// TIA Portal V19 export
FUNCTION_BLOCK "ButtonsSafe_LB211"   // FB167, LAD
TITLE = LB211 SAFE BUTTONS (@Rollformer) used for feed Area 02 material
// stored: MemoryReserve 100, SetENOAutomatically false
   VAR_INPUT
      Reset_OthersPBs_Activation_IN : Bool := FALSE;
   END_VAR
   VAR_OUTPUT
      Reset_OthersPBs_Activation_OUT : Bool;
   END_VAR
   VAR
      SelectionIs_Bwd : Bool;
      SelectionIs_Fwd : Bool;
      Pb_PEAux : Bool;
      PB : Struct
         ResetAlarms : Bool;
         Rollformer_Bwd : Bool;
         Rollformer_Fwd : Bool;
      END_STRUCT;
   END_VAR
   VAR_TEMP
      EnablingSwitch : Bool;
      Pb_PositiveEdge : Bool;
   END_VAR
   VAR_TEMP   // added for the SCL form of the ladder/FBD networks
      _w1 : Bool;
   END_VAR
BEGIN

REGION Network 1: Enabling switch positive edge
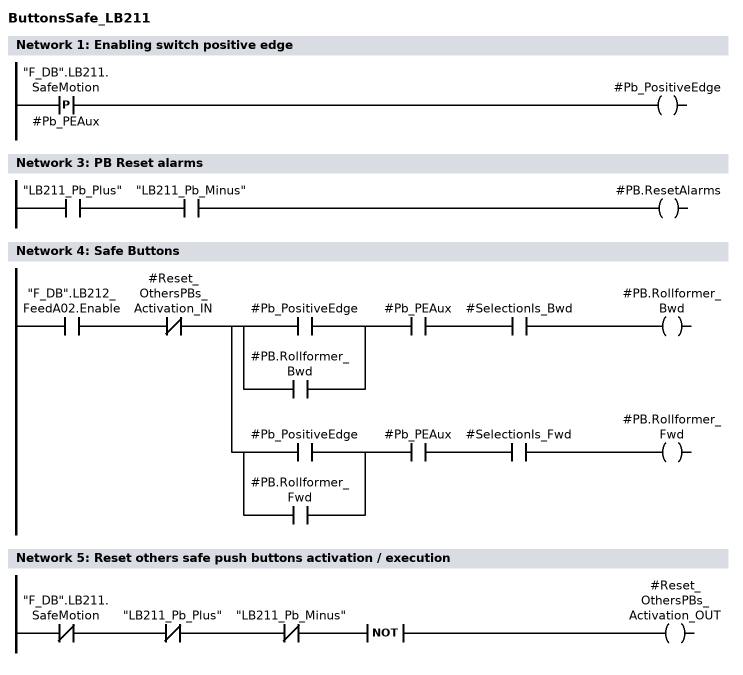
   RUNG wire#powerrail
      P_Contact(operand := "F_DB".LB211.SafeMotion, bit := #Pb_PEAux)
      Coil( #Pb_PositiveEdge )
   END_RUNG
   // the same network as SCL:
   #_w1 := "F_DB".LB211.SafeMotion AND NOT #Pb_PEAux;   // rising edge of "F_DB".LB211.SafeMotion
   #Pb_PEAux := "F_DB".LB211.SafeMotion;
   #Pb_PositiveEdge := #_w1;
END_REGION

REGION Network 2 (SCL): Selection of direction

   IF "LB211_Pb_Plus" AND  "LB211_Pb_Minus" THEN
       #SelectionIs_Fwd := FALSE;
       #SelectionIs_Bwd := FALSE;

   ELSIF "F_DB".LB211.SafeMotion THEN
       ;

   ELSIF "LB211_Pb_Plus" AND NOT "LB211_Pb_Minus"  THEN
       #SelectionIs_Fwd := TRUE;
       #SelectionIs_Bwd := FALSE;

   ELSIF "LB211_Pb_Minus" AND NOT "LB211_Pb_Plus" THEN
       #SelectionIs_Bwd := TRUE;       
       #SelectionIs_Fwd := FALSE;  
   END_IF;
END_REGION

REGION Network 3: PB Reset alarms
   RUNG wire#powerrail
      Contact( "LB211_Pb_Plus" )
      Contact( "LB211_Pb_Minus" )
      Coil( #PB.ResetAlarms )
   END_RUNG
   // the same network as SCL:
   #PB.ResetAlarms := "LB211_Pb_Plus" AND "LB211_Pb_Minus";
END_REGION

REGION Network 4: Safe Buttons
   RUNG wire#powerrail
      Contact( "F_DB".LB212_FeedA02.Enable )
      I_Contact( #Reset_OthersPBs_Activation_IN )
      wire#w1
      Contact( #Pb_PositiveEdge )
      wire#w2
      Contact( #Pb_PEAux )
      Contact( #SelectionIs_Bwd )
      Coil( #PB.Rollformer_Bwd )
   END_RUNG
   RUNG wire#w1
      Contact( #PB.Rollformer_Bwd )
   END_RUNG wire#w2
   RUNG wire#w1
      Contact( #Pb_PositiveEdge )
      wire#w3
      Contact( #Pb_PEAux )
      Contact( #SelectionIs_Fwd )
      Coil( #PB.Rollformer_Fwd )
   END_RUNG
   RUNG wire#w1
      Contact( #PB.Rollformer_Fwd )
   END_RUNG wire#w3
   // the same network as SCL:
   #_w1 := "F_DB".LB212_FeedA02.Enable AND NOT #Reset_OthersPBs_Activation_IN;
   #PB.Rollformer_Bwd := #_w1 AND (#Pb_PositiveEdge OR #PB.Rollformer_Bwd) AND #Pb_PEAux AND #SelectionIs_Bwd;
   #PB.Rollformer_Fwd := #_w1 AND (#Pb_PositiveEdge OR #PB.Rollformer_Fwd) AND #Pb_PEAux AND #SelectionIs_Fwd;
END_REGION

REGION Network 5: Reset others safe push buttons activation / execution
   RUNG wire#powerrail
      I_Contact( "F_DB".LB211.SafeMotion )
      I_Contact( "LB211_Pb_Plus" )
      I_Contact( "LB211_Pb_Minus" )
      Not()
      Coil( #Reset_OthersPBs_Activation_OUT )
   END_RUNG
   // the same network as SCL:
   #Reset_OthersPBs_Activation_OUT := NOT (NOT "F_DB".LB211.SafeMotion AND NOT "LB211_Pb_Plus" AND NOT "LB211_Pb_Minus");
END_REGION

REGION Network 6: >
END_REGION

REGION Network 7: >
END_REGION

REGION Network 8: >
END_REGION
END_FUNCTION_BLOCK
